# EPICS autosave request: ipApp/Db/JenaNV40_settings.req
# Jena NV40/1CLE
$(P)$(C)write
$(P)$(C)write.PREC
$(P)$(C)read.DESC
$(P)$(C)read.PREC
$(P)$(C)read.SCAN
$(P)$(C)cl
$(P)$(C)rc
